FUNCTION_BLOCK Load
  (* Standard: 61499-2 *)
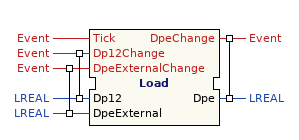
  EVENT_INPUT
    Tick;
    Dp12Change WITH Dp12;
    DpeExternalChange WITH DpeExternal;
  END_EVENT
  EVENT_OUTPUT
    DpeChange WITH Dpe;
  END_EVENT
  VAR_INPUT
    Dp12 : LREAL;
    DpeExternal : LREAL := 0;
  END_VAR
  VAR_OUTPUT
    Dpe : LREAL;
  END_VAR
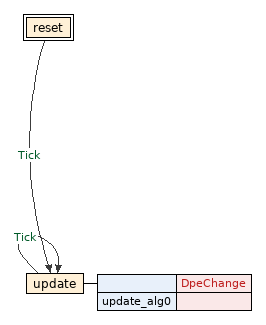
  EC_STATES
    reset;
    update : -> DpeChange, update_alg0;
  END_STATES
  EC_TRANSITIONS
    reset TO update := Tick;
    update TO update := Tick;
  END_TRANSITIONS
  ALGORITHM update_alg0 IN ST:
Dpe := Dp12 + DpeExternal;
  END_ALGORITHM
END_FUNCTION_BLOCK
